INTERFACE I_ArrayDatatypeAddedEvent EXTENDS I_Event

PROPERTY PUBLIC Target : I_ArrayDatatype
GET
END_GET
END_PROPERTY

END_INTERFACE

(* stored: Version 1.1.0.1, ProductVersion 3.1.4024.13
   Itf I_ArrayDatatypeAddedEvent: Id {5a140093-2486-0e7c-3a88-fa72b434e184}
   Property Target: Id {ffb525d3-ca53-053a-3cb5-14c342254a0c}
   Get Get: Id {789781b9-6d29-02bb-165d-025716045142} *)
